// TIA Portal V20 export
DATA_BLOCK "SBK11"   // DB324
// stored: MemoryReserve 100
   VAR
      "GATE EC SCRAP BOX-2 PB.LOCK" : Bool := FALSE;
      "GATE EC SCRAP BOX-2 PB.RESET" : Bool := FALSE;
      SPARE : Bool := FALSE;
      SPARE_1 : Bool := FALSE;
      "GATE EC SCRAP BOX-2 PB.UNLOCK" : Bool := FALSE;
      SPARE_2 : Bool := FALSE;
      SPARE_3 : Bool := FALSE;
      SPARE_4 : Bool := FALSE;
      "GATE EC SCRAP BOX-2 PL.LOCK" : Bool := FALSE;
      "GATE EC SCRAP BOX-2 PL.UNLOCK" : Bool := TRUE;
      "GATE EC SCRAP BOX-2 PL.RESET" : Bool := FALSE;
   END_VAR
BEGIN
END_DATA_BLOCK
